ABB RAPID module: Module1.mod

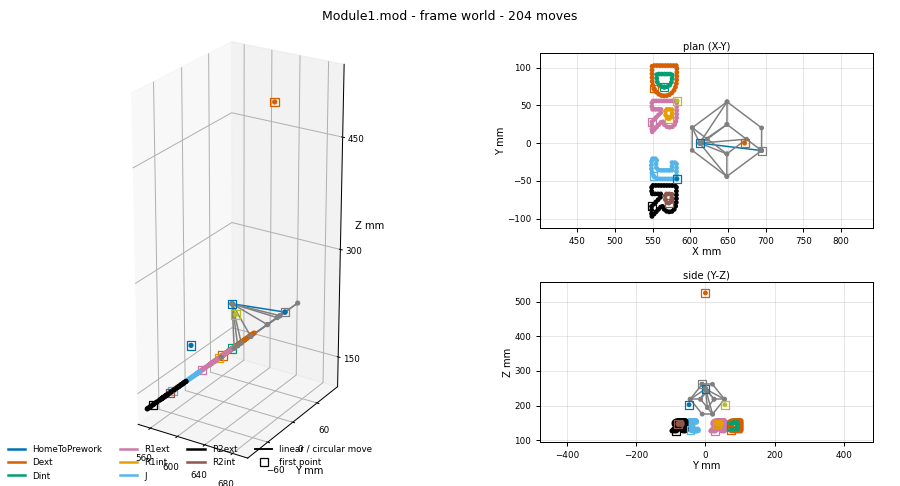
[picture p0: tool path of Module1.mod in frame world, 204 of 204 moves have a stored position in this frame; points joined in program order, loops and branches not executed]
MODULE Module1
    PERS tooldata MyNewTool:=[TRUE,[[40,0,140],[1,0,0,0]],[0.2,[0,0,1],[1,0,0,0],0,0,0]];
    PERS tooldata MaRCK:=[TRUE,[[40,0,140],[1,0,0,0]],[1,[0,0,60],[1,0,0,0],0,0,0]];
    PERS tooldata Marcket:=[TRUE,[[40,0,140],[1,0,0,0]],[1,[0,0,1],[1,0,0,0],0,0,0]];
    CONST robtarget PreworkLogo:=[[612.590636345,0.112352276,247.897245036],[0.173647946,0.001613761,0.984806431,-0.000284548],[-1,0,0,0],[9E+09,9E+09,9E+09,9E+09,9E+09,9E+09]];
    CONST robtarget EDext_10:=[[551.912875252,72.53519352,128.929412083],[0.173647946,0.001613761,0.984806431,-0.000284548],[0,-2,1,0],[9E+09,9E+09,9E+09,9E+09,9E+09,9E+09]];
    CONST robtarget EDext_20:=[[550.351593621,77.035190099,127.453730912],[0.173647946,0.001613761,0.984806431,-0.000284548],[0,0,0,0],[9E+09,9E+09,9E+09,9E+09,9E+09,9E+09]];
    CONST robtarget EDext_30:=[[549.633220287,81.925977855,126.766089465],[0.173647946,0.001613761,0.984806431,-0.000284548],[0,0,0,0],[9E+09,9E+09,9E+09,9E+09,9E+09,9E+09]];
    CONST robtarget EDext_40:=[[549.374310427,86.910926647,126.508367741],[0.173647946,0.001613761,0.984806431,-0.000284548],[0,0,0,0],[9E+09,9E+09,9E+09,9E+09,9E+09,9E+09]];
    CONST robtarget EDext_50:=[[549.36766375,91.910642603,126.486801869],[0.173647946,0.001613761,0.984806431,-0.000284548],[0,0,0,0],[9E+09,9E+09,9E+09,9E+09,9E+09,9E+09]];
    CONST robtarget EDext_60:=[[549.384050297,96.910615751,126.486801869],[0.173647946,0.001613761,0.984806431,-0.000284548],[0,0,0,0],[9E+09,9E+09,9E+09,9E+09,9E+09,9E+09]];
    CONST robtarget EDext_70:=[[549.400436844,101.910588899,126.486801869],[0.173647946,0.001613761,0.984806431,-0.000284548],[0,0,0,0],[9E+09,9E+09,9E+09,9E+09,9E+09,9E+09]];
    CONST robtarget EDext_80:=[[552.263411146,102.983965117,129.164192022],[0.173647946,0.001613761,0.984806431,-0.000284548],[0,0,0,0],[9E+09,9E+09,9E+09,9E+09,9E+09,9E+09]];
    CONST robtarget EDext_90:=[[555.913201428,102.97200356,132.581630802],[0.173647946,0.001613761,0.984806431,-0.000284548],[0,0,0,0],[9E+09,9E+09,9E+09,9E+09,9E+09,9E+09]];
    CONST robtarget EDext_100:=[[559.562991711,102.960042004,135.999069582],[0.173647946,0.001613761,0.984806431,-0.000284548],[0,0,0,0],[9E+09,9E+09,9E+09,9E+09,9E+09,9E+09]];
    CONST robtarget EDext_110:=[[563.212781993,102.948080447,139.416508362],[0.173647946,0.001613761,0.984806431,-0.000284548],[0,0,0,0],[9E+09,9E+09,9E+09,9E+09,9E+09,9E+09]];
    CONST robtarget EDext_120:=[[566.862572275,102.936118891,142.833947142],[0.173647946,0.001613761,0.984806431,-0.000284548],[0,0,0,0],[9E+09,9E+09,9E+09,9E+09,9E+09,9E+09]];
    CONST robtarget EDext_130:=[[570.512362558,102.924157334,146.251385922],[0.173647946,0.001613761,0.984806431,-0.000284548],[0,0,0,0],[9E+09,9E+09,9E+09,9E+09,9E+09,9E+09]];
    CONST robtarget EDext_140:=[[574.16215284,102.912195777,149.668824701],[0.173647946,0.001613761,0.984806431,-0.000284548],[0,0,0,0],[9E+09,9E+09,9E+09,9E+09,9E+09,9E+09]];
    CONST robtarget EDext_150:=[[577.811943123,102.900234221,153.086263481],[0.173647946,0.001613761,0.984806431,-0.000284548],[0,0,0,0],[9E+09,9E+09,9E+09,9E+09,9E+09,9E+09]];
    CONST robtarget EDext_160:=[[581.461733405,102.888272664,156.503702261],[0.173647946,0.001613761,0.984806431,-0.000284548],[0,0,0,0],[9E+09,9E+09,9E+09,9E+09,9E+09,9E+09]];
    CONST robtarget EDext_170:=[[582.239259874,98.968456724,157.243750889],[0.173647946,0.001613761,0.984806431,-0.000284548],[0,0,0,0],[9E+09,9E+09,9E+09,9E+09,9E+09,9E+09]];
    CONST robtarget EDext_180:=[[582.222873327,93.968483576,157.243750889],[0.173647946,0.001613761,0.984806431,-0.000284548],[0,0,0,0],[9E+09,9E+09,9E+09,9E+09,9E+09,9E+09]];
    CONST robtarget EDext_190:=[[582.206486779,88.968510428,157.243750889],[0.173647946,0.001613761,0.984806431,-0.000284548],[0,0,0,0],[9E+09,9E+09,9E+09,9E+09,9E+09,9E+09]];
    CONST robtarget EDext_200:=[[582.05998145,83.973285517,157.121902414],[0.173647946,0.001613761,0.984806431,-0.000284548],[0,0,0,0],[9E+09,9E+09,9E+09,9E+09,9E+09,9E+09]];
    CONST robtarget EDext_210:=[[581.599769178,79.014590704,156.706209142],[0.173647946,0.001613761,0.984806431,-0.000284548],[0,0,0,0],[9E+09,9E+09,9E+09,9E+09,9E+09,9E+09]];
    CONST robtarget EDext_220:=[[580.404388174,74.301796937,155.601401967],[0.173647946,0.001613761,0.984806431,-0.000284548],[0,0,0,0],[9E+09,9E+09,9E+09,9E+09,9E+09,9E+09]];
    CONST robtarget EDext_230:=[[578.391013182,70.140860724,153.728990378],[0.173647946,0.001613761,0.984806431,-0.000284548],[0,0,0,0],[9E+09,9E+09,9E+09,9E+09,9E+09,9E+09]];
    CONST robtarget EDext_240:=[[575.690696414,66.788466394,151.210894602],[0.173647946,0.001613761,0.984806431,-0.000284548],[0,0,0,0],[9E+09,9E+09,9E+09,9E+09,9E+09,9E+09]];
    CONST robtarget EDext_250:=[[572.487460802,64.407050959,148.218922062],[0.173647946,0.001613761,0.984806431,-0.000284548],[0,0,0,0],[9E+09,9E+09,9E+09,9E+09,9E+09,9E+09]];
    CONST robtarget EDext_260:=[[568.966787181,63.118163403,144.926370726],[0.173647946,0.001613761,0.984806431,-0.000284548],[0,0,0,0],[9E+09,9E+09,9E+09,9E+09,9E+09,9E+09]];
    CONST robtarget EDext_270:=[[565.328580893,62.794822032,141.520807298],[0.173647946,0.001613761,0.984806431,-0.000284548],[0,0,0,0],[9E+09,9E+09,9E+09,9E+09,9E+09,9E+09]];
    CONST robtarget EDext_280:=[[561.709530664,63.365475702,138.130436868],[0.173647946,0.001613761,0.984806431,-0.000284548],[0,0,0,0],[9E+09,9E+09,9E+09,9E+09,9E+09,9E+09]];
    CONST robtarget EDext_290:=[[558.268704982,64.989283235,134.903711368],[0.173647946,0.001613761,0.984806431,-0.000284548],[0,0,0,0],[9E+09,9E+09,9E+09,9E+09,9E+09,9E+09]];
    CONST robtarget EDext_300:=[[555.180659774,67.628712266,132.004187631],[0.173647946,0.001613761,0.984806431,-0.000284548],[0,0,0,0],[9E+09,9E+09,9E+09,9E+09,9E+09,9E+09]];
    CONST robtarget EDext_310:=[[552.613212389,71.156303357,129.589388927],[0.173647946,0.001613761,0.984806431,-0.000284548],[0,0,0,0],[9E+09,9E+09,9E+09,9E+09,9E+09,9E+09]];
    CONST robtarget FDint_10:=[[565.761082243,74.386090886,141.890200973],[0.173647946,0.001613761,0.984806431,-0.000284548],[0,-2,1,0],[9E+09,9E+09,9E+09,9E+09,9E+09,9E+09]];
    CONST robtarget FDint_20:=[[569.379445273,74.944551838,145.276463096],[0.173647946,0.001613761,0.984806431,-0.000284548],[0,0,0,0],[9E+09,9E+09,9E+09,9E+09,9E+09,9E+09]];
    CONST robtarget FDint_30:=[[572.681520952,77.008685984,148.361956019],[0.173647946,0.001613761,0.984806431,-0.000284548],[0,0,0,0],[9E+09,9E+09,9E+09,9E+09,9E+09,9E+09]];
    CONST robtarget FDint_40:=[[575.047866711,80.768438651,150.566095233],[0.173647946,0.001613761,0.984806431,-0.000284548],[0,0,0,0],[9E+09,9E+09,9E+09,9E+09,9E+09,9E+09]];
    CONST robtarget FDint_50:=[[575.986682219,85.560327407,151.430430149],[0.173647946,0.001613761,0.984806431,-0.000284548],[0,0,0,0],[9E+09,9E+09,9E+09,9E+09,9E+09,9E+09]];
    CONST robtarget FDint_60:=[[576.087876515,90.558290854,151.509844214],[0.173647946,0.001613761,0.984806431,-0.000284548],[0,0,0,0],[9E+09,9E+09,9E+09,9E+09,9E+09,9E+09]];
    CONST robtarget FDint_70:=[[573.20406064,91.610574886,148.806416589],[0.173647946,0.001613761,0.984806431,-0.000284548],[0,0,0,0],[9E+09,9E+09,9E+09,9E+09,9E+09,9E+09]];
    CONST robtarget FDint_80:=[[569.554270358,91.622536443,145.388977809],[0.173647946,0.001613761,0.984806431,-0.000284548],[0,0,0,0],[9E+09,9E+09,9E+09,9E+09,9E+09,9E+09]];
    CONST robtarget FDint_90:=[[565.904480074,91.634497999,141.971539029],[0.173647946,0.001613761,0.984806431,-0.000284548],[0,0,0,0],[9E+09,9E+09,9E+09,9E+09,9E+09,9E+09]];
    CONST robtarget FDint_100:=[[562.254689792,91.646459556,138.554100249],[0.173647946,0.001613761,0.984806431,-0.000284548],[0,0,0,0],[9E+09,9E+09,9E+09,9E+09,9E+09,9E+09]];
    CONST robtarget FDint_110:=[[558.604899509,91.658421112,135.136661469],[0.173647946,0.001613761,0.984806431,-0.000284548],[0,0,0,0],[9E+09,9E+09,9E+09,9E+09,9E+09,9E+09]];
    CONST robtarget FDint_120:=[[555.51395758,90.900193665,132.244851682],[0.173647946,0.001613761,0.984806431,-0.000284548],[0,0,0,0],[9E+09,9E+09,9E+09,9E+09,9E+09,9E+09]];
    CONST robtarget FDint_130:=[[555.56318478,85.901073737,132.306285076],[0.173647946,0.001613761,0.984806431,-0.000284548],[0,0,0,0],[9E+09,9E+09,9E+09,9E+09,9E+09,9E+09]];
    CONST robtarget FDint_140:=[[556.34730194,81.067926581,133.055307452],[0.173647946,0.001613761,0.984806431,-0.000284548],[0,0,0,0],[9E+09,9E+09,9E+09,9E+09,9E+09,9E+09]];
    CONST robtarget FDint_150:=[[558.624417237,77.220561783,135.199241268],[0.173647946,0.001613761,0.984806431,-0.000284548],[0,0,0,0],[9E+09,9E+09,9E+09,9E+09,9E+09,9E+09]];
    CONST robtarget FDint_160:=[[561.87847136,75.038381865,138.252800717],[0.173647946,0.001613761,0.984806431,-0.000284548],[0,0,0,0],[9E+09,9E+09,9E+09,9E+09,9E+09,9E+09]];
    CONST robtarget FDint_170:=[[565.486835279,74.389591817,141.633405025],[0.173647946,0.001613761,0.984806431,-0.000284548],[0,0,0,0],[9E+09,9E+09,9E+09,9E+09,9E+09,9E+09]];
    CONST robtarget GR1ext_10:=[[549.159222937,28.309785163,126.486801869],[0.173647946,0.001613761,0.984806431,-0.000284548],[0,0,0,0],[9E+09,9E+09,9E+09,9E+09,9E+09,9E+09]];
    CONST robtarget GR1ext_20:=[[552.078895967,31.318504465,129.211341749],[0.173647946,0.001613761,0.984806431,-0.000284548],[0,0,0,0],[9E+09,9E+09,9E+09,9E+09,9E+09,9E+09]];
    CONST robtarget GR1ext_30:=[[554.998568997,34.327223766,131.93588163],[0.173647946,0.001613761,0.984806431,-0.000284548],[0,0,0,0],[9E+09,9E+09,9E+09,9E+09,9E+09,9E+09]];
    CONST robtarget GR1ext_40:=[[557.918242027,37.335943068,134.660421511],[0.173647946,0.001613761,0.984806431,-0.000284548],[0,0,0,0],[9E+09,9E+09,9E+09,9E+09,9E+09,9E+09]];
    CONST robtarget GR1ext_50:=[[560.837915058,40.344662369,137.384961391],[0.173647946,0.001613761,0.984806431,-0.000284548],[0,0,0,0],[9E+09,9E+09,9E+09,9E+09,9E+09,9E+09]];
    CONST robtarget GR1ext_60:=[[561.129703813,44.863025586,137.644306177],[0.173647946,0.001613761,0.984806431,-0.000284548],[0,0,0,0],[9E+09,9E+09,9E+09,9E+09,9E+09,9E+09]];
    CONST robtarget GR1ext_70:=[[557.47991353,44.874987143,134.226867398],[0.173647946,0.001613761,0.984806431,-0.000284548],[0,0,0,0],[9E+09,9E+09,9E+09,9E+09,9E+09,9E+09]];
    CONST robtarget GR1ext_80:=[[553.830123248,44.886948699,130.809428618],[0.173647946,0.001613761,0.984806431,-0.000284548],[0,0,0,0],[9E+09,9E+09,9E+09,9E+09,9E+09,9E+09]];
    CONST robtarget GR1ext_90:=[[550.180332966,44.898910256,127.391989838],[0.173647946,0.001613761,0.984806431,-0.000284548],[0,0,0,0],[9E+09,9E+09,9E+09,9E+09,9E+09,9E+09]];
    CONST robtarget GR1ext_100:=[[549.2256475,48.577692778,126.486801869],[0.173647946,0.001613761,0.984806431,-0.000284548],[0,0,0,0],[9E+09,9E+09,9E+09,9E+09,9E+09,9E+09]];
    CONST robtarget GR1ext_110:=[[549.242034047,53.577665926,126.486801869],[0.173647946,0.001613761,0.984806431,-0.000284548],[0,0,0,0],[9E+09,9E+09,9E+09,9E+09,9E+09,9E+09]];
    CONST robtarget GR1ext_120:=[[551.034331948,56.127938354,128.157155282],[0.173647946,0.001613761,0.984806431,-0.000284548],[0,0,0,0],[9E+09,9E+09,9E+09,9E+09,9E+09,9E+09]];
    CONST robtarget GR1ext_130:=[[554.68412223,56.115976798,131.574594062],[0.173647946,0.001613761,0.984806431,-0.000284548],[0,0,0,0],[9E+09,9E+09,9E+09,9E+09,9E+09,9E+09]];
    CONST robtarget GR1ext_140:=[[558.333912513,56.104015241,134.992032842],[0.173647946,0.001613761,0.984806431,-0.000284548],[0,0,0,0],[9E+09,9E+09,9E+09,9E+09,9E+09,9E+09]];
    CONST robtarget GR1ext_150:=[[561.983702796,56.092053685,138.409471622],[0.173647946,0.001613761,0.984806431,-0.000284548],[0,0,0,0],[9E+09,9E+09,9E+09,9E+09,9E+09,9E+09]];
    CONST robtarget GR1ext_160:=[[565.633493078,56.080092128,141.826910402],[0.173647946,0.001613761,0.984806431,-0.000284548],[0,0,0,0],[9E+09,9E+09,9E+09,9E+09,9E+09,9E+09]];
    CONST robtarget GR1ext_170:=[[569.283283361,56.068130572,145.244349182],[0.173647946,0.001613761,0.984806431,-0.000284548],[0,0,0,0],[9E+09,9E+09,9E+09,9E+09,9E+09,9E+09]];
    CONST robtarget GR1ext_180:=[[572.933073643,56.056169015,148.661787962],[0.173647946,0.001613761,0.984806431,-0.000284548],[0,0,0,0],[9E+09,9E+09,9E+09,9E+09,9E+09,9E+09]];
    CONST robtarget GR1ext_190:=[[576.582863926,56.044207459,152.079226742],[0.173647946,0.001613761,0.984806431,-0.000284548],[0,0,0,0],[9E+09,9E+09,9E+09,9E+09,9E+09,9E+09]];
    CONST robtarget GR1ext_200:=[[580.232654208,56.032245902,155.496665522],[0.173647946,0.001613761,0.984806431,-0.000284548],[0,0,0,0],[9E+09,9E+09,9E+09,9E+09,9E+09,9E+09]];
    CONST robtarget GR1ext_210:=[[582.090514517,53.582276609,157.243750889],[0.173647946,0.001613761,0.984806431,-0.000284548],[0,0,0,0],[9E+09,9E+09,9E+09,9E+09,9E+09,9E+09]];
    CONST robtarget GR1ext_220:=[[582.07412797,48.582303461,157.243750889],[0.173647946,0.001613761,0.984806431,-0.000284548],[0,0,0,0],[9E+09,9E+09,9E+09,9E+09,9E+09,9E+09]];
    CONST robtarget GR1ext_230:=[[582.057741422,43.582330312,157.243750889],[0.173647946,0.001613761,0.984806431,-0.000284548],[0,0,0,0],[9E+09,9E+09,9E+09,9E+09,9E+09,9E+09]];
    CONST robtarget GR1ext_240:=[[582.041354875,38.582357164,157.243750889],[0.173647946,0.001613761,0.984806431,-0.000284548],[0,0,0,0],[9E+09,9E+09,9E+09,9E+09,9E+09,9E+09]];
    CONST robtarget GR1ext_250:=[[581.887031,33.588566956,157.114577286],[0.173647946,0.001613761,0.984806431,-0.000284548],[0,0,0,0],[9E+09,9E+09,9E+09,9E+09,9E+09,9E+09]];
    CONST robtarget GR1ext_260:=[[581.128662004,28.711829147,156.419459926],[0.173647946,0.001613761,0.984806431,-0.000284548],[0,0,0,0],[9E+09,9E+09,9E+09,9E+09,9E+09,9E+09]];
    CONST robtarget GR1ext_270:=[[579.222937052,24.480084612,154.648061408],[0.173647946,0.001613761,0.984806431,-0.000284548],[0,0,0,0],[9E+09,9E+09,9E+09,9E+09,9E+09,9E+09]];
    CONST robtarget GR1ext_280:=[[576.214714314,21.722189391,151.839840233],[0.173647946,0.001613761,0.984806431,-0.000284548],[0,0,0,0],[9E+09,9E+09,9E+09,9E+09,9E+09,9E+09]];
    CONST robtarget GR1ext_290:=[[572.616939057,21.053869541,148.473192144],[0.173647946,0.001613761,0.984806431,-0.000284548],[0,0,0,0],[9E+09,9E+09,9E+09,9E+09,9E+09,9E+09]];
    CONST robtarget GR1ext_300:=[[569.03162427,21.867677864,145.113663007],[0.173647946,0.001613761,0.984806431,-0.000284548],[0,0,0,0],[9E+09,9E+09,9E+09,9E+09,9E+09,9E+09]];
    CONST robtarget GR1ext_310:=[[565.933301553,24.431725119,142.204747469],[0.173647946,0.001613761,0.984806431,-0.000284548],[0,0,0,0],[9E+09,9E+09,9E+09,9E+09,9E+09,9E+09]];
    CONST robtarget GR1ext_320:=[[563.657751182,28.309232507,140.062186439],[0.173647946,0.001613761,0.984806431,-0.000284548],[0,0,0,0],[9E+09,9E+09,9E+09,9E+09,9E+09,9E+09]];
    CONST robtarget GR1ext_330:=[[561.138391327,27.497607501,137.705729007],[0.173647946,0.001613761,0.984806431,-0.000284548],[0,0,0,0],[9E+09,9E+09,9E+09,9E+09,9E+09,9E+09]];
    CONST robtarget GR1ext_340:=[[558.264968647,24.406364665,135.024747876],[0.173647946,0.001613761,0.984806431,-0.000284548],[0,0,0,0],[9E+09,9E+09,9E+09,9E+09,9E+09,9E+09]];
    CONST robtarget GR1ext_350:=[[555.391545966,21.315121829,132.343766744],[0.173647946,0.001613761,0.984806431,-0.000284548],[0,0,0,0],[9E+09,9E+09,9E+09,9E+09,9E+09,9E+09]];
    CONST robtarget GR1ext_360:=[[552.518123285,18.223878993,129.662785613],[0.173647946,0.001613761,0.984806431,-0.000284548],[0,0,0,0],[9E+09,9E+09,9E+09,9E+09,9E+09,9E+09]];
    CONST robtarget GR1ext_370:=[[549.644700604,15.132636157,126.981804481],[0.173647946,0.001613761,0.984806431,-0.000284548],[0,0,0,0],[9E+09,9E+09,9E+09,9E+09,9E+09,9E+09]];
    CONST robtarget GR1ext_380:=[[549.127527591,18.638688665,126.486801869],[0.173647946,0.001613761,0.984806431,-0.000284548],[0,0,0,0],[9E+09,9E+09,9E+09,9E+09,9E+09,9E+09]];
    CONST robtarget GR1ext_390:=[[549.143914138,23.638661813,126.486801869],[0.173647946,0.001613761,0.984806431,-0.000284548],[0,0,0,0],[9E+09,9E+09,9E+09,9E+09,9E+09,9E+09]];
    CONST robtarget HR1int_10:=[[571.959732893,32.647563873,147.822254349],[0.173647946,0.001613761,0.984806431,-0.000284548],[0,-2,1,0],[9E+09,9E+09,9E+09,9E+09,9E+09,9E+09]];
    CONST robtarget HR1int_20:=[[575.149419403,34.61134025,150.802822071],[0.173647946,0.001613761,0.984806431,-0.000284548],[0,0,0,0],[9E+09,9E+09,9E+09,9E+09,9E+09,9E+09]];
    CONST robtarget HR1int_30:=[[575.982626554,39.413197479,151.5682423],[0.173647946,0.001613761,0.984806431,-0.000284548],[0,0,0,0],[9E+09,9E+09,9E+09,9E+09,9E+09,9E+09]];
    CONST robtarget HR1int_40:=[[576.017836302,44.412828089,151.585868046],[0.173647946,0.001613761,0.984806431,-0.000284548],[0,0,0,0],[9E+09,9E+09,9E+09,9E+09,9E+09,9E+09]];
    CONST robtarget HR1int_50:=[[572.662368207,44.825229273,148.442782661],[0.173647946,0.001613761,0.984806431,-0.000284548],[0,0,0,0],[9E+09,9E+09,9E+09,9E+09,9E+09,9E+09]];
    CONST robtarget HR1int_60:=[[569.012577925,44.83719083,145.025343881],[0.173647946,0.001613761,0.984806431,-0.000284548],[0,0,0,0],[9E+09,9E+09,9E+09,9E+09,9E+09,9E+09]];
    CONST robtarget HR1int_70:=[[567.17340627,42.351576284,143.310902832],[0.173647946,0.001613761,0.984806431,-0.000284548],[0,0,0,0],[9E+09,9E+09,9E+09,9E+09,9E+09,9E+09]];
    CONST robtarget HR1int_80:=[[567.402598455,37.370563966,143.540786974],[0.173647946,0.001613761,0.984806431,-0.000284548],[0,0,0,0],[9E+09,9E+09,9E+09,9E+09,9E+09,9E+09]];
    CONST robtarget HR1int_90:=[[569.422495165,33.396346001,145.444269007],[0.173647946,0.001613761,0.984806431,-0.000284548],[0,0,0,0],[9E+09,9E+09,9E+09,9E+09,9E+09,9E+09]];
    CONST robtarget IJ_10:=[[551.320468068,-43.245490091,128.730015331],[0.173647946,0.001613761,0.984806431,-0.000284548],[0,0,0,0],[9E+09,9E+09,9E+09,9E+09,9E+09,9E+09]];
    CONST robtarget IJ_20:=[[549.426005203,-39.008514231,126.943174249],[0.173647946,0.001613761,0.984806431,-0.000284548],[0,0,0,0],[9E+09,9E+09,9E+09,9E+09,9E+09,9E+09]];
    CONST robtarget IJ_30:=[[548.586005622,-34.15957373,126.141779114],[0.173647946,0.001613761,0.984806431,-0.000284548],[0,0,0,0],[9E+09,9E+09,9E+09,9E+09,9E+09,9E+09]];
    CONST robtarget IJ_40:=[[548.477427418,-29.166511841,126.024792284],[0.173647946,0.001613761,0.984806431,-0.000284548],[0,0,0,0],[9E+09,9E+09,9E+09,9E+09,9E+09,9E+09]];
    CONST robtarget IJ_50:=[[548.710119201,-24.177436392,126.227358447],[0.173647946,0.001613761,0.984806431,-0.000284548],[0,0,0,0],[9E+09,9E+09,9E+09,9E+09,9E+09,9E+09]];
    CONST robtarget IJ_60:=[[550.104401144,-20.559048954,127.521760564],[0.173647946,0.001613761,0.984806431,-0.000284548],[0,0,0,0],[9E+09,9E+09,9E+09,9E+09,9E+09,9E+09]];
    CONST robtarget IJ_70:=[[553.754191426,-20.57101051,130.939199344],[0.173647946,0.001613761,0.984806431,-0.000284548],[0,0,0,0],[9E+09,9E+09,9E+09,9E+09,9E+09,9E+09]];
    CONST robtarget IJ_80:=[[555.465361118,-22.711275868,132.547983754],[0.173647946,0.001613761,0.984806431,-0.000284548],[0,0,0,0],[9E+09,9E+09,9E+09,9E+09,9E+09,9E+09]];
    CONST robtarget IJ_90:=[[554.680121136,-27.565791663,131.827638136],[0.173647946,0.001613761,0.984806431,-0.000284548],[0,0,0,0],[9E+09,9E+09,9E+09,9E+09,9E+09,9E+09]];
    CONST robtarget IJ_100:=[[555.145862124,-32.487268808,132.278826933],[0.173647946,0.001613761,0.984806431,-0.000284548],[0,0,0,0],[9E+09,9E+09,9E+09,9E+09,9E+09,9E+09]];
    CONST robtarget IJ_110:=[[557.841723431,-35.563111404,134.812476972],[0.173647946,0.001613761,0.984806431,-0.000284548],[0,0,0,0],[9E+09,9E+09,9E+09,9E+09,9E+09,9E+09]];
    CONST robtarget IJ_120:=[[561.46746702,-35.976374681,138.208631607],[0.173647946,0.001613761,0.984806431,-0.000284548],[0,0,0,0],[9E+09,9E+09,9E+09,9E+09,9E+09,9E+09]];
    CONST robtarget IJ_130:=[[565.117207108,-35.997312406,141.626050933],[0.173647946,0.001613761,0.984806431,-0.000284548],[0,0,0,0],[9E+09,9E+09,9E+09,9E+09,9E+09,9E+09]];
    CONST robtarget IJ_140:=[[568.766997391,-36.009273962,145.043489713],[0.173647946,0.001613761,0.984806431,-0.000284548],[0,0,0,0],[9E+09,9E+09,9E+09,9E+09,9E+09,9E+09]];
    CONST robtarget IJ_150:=[[572.416787673,-36.021235519,148.460928493],[0.173647946,0.001613761,0.984806431,-0.000284548],[0,0,0,0],[9E+09,9E+09,9E+09,9E+09,9E+09,9E+09]];
    CONST robtarget IJ_160:=[[575.835093356,-35.713886099,151.660641828],[0.173647946,0.001613761,0.984806431,-0.000284548],[0,0,0,0],[9E+09,9E+09,9E+09,9E+09,9E+09,9E+09]];
    CONST robtarget IJ_170:=[[575.851479904,-30.713912951,151.660641828],[0.173647946,0.001613761,0.984806431,-0.000284548],[0,0,0,0],[9E+09,9E+09,9E+09,9E+09,9E+09,9E+09]];
    CONST robtarget IJ_180:=[[575.893242248,-25.7489433,151.68450932],[0.173647946,0.001613761,0.984806431,-0.000284548],[0,0,0,0],[9E+09,9E+09,9E+09,9E+09,9E+09,9E+09]];
    CONST robtarget IJ_190:=[[579.543032531,-25.760904857,155.1019481],[0.173647946,0.001613761,0.984806431,-0.000284548],[0,0,0,0],[9E+09,9E+09,9E+09,9E+09,9E+09,9E+09]];
    CONST robtarget IJ_200:=[[581.824339743,-27.634754078,157.243750889],[0.173647946,0.001613761,0.984806431,-0.000284548],[0,0,0,0],[9E+09,9E+09,9E+09,9E+09,9E+09,9E+09]];
    CONST robtarget IJ_210:=[[581.807953196,-32.634727226,157.243750889],[0.173647946,0.001613761,0.984806431,-0.000284548],[0,0,0,0],[9E+09,9E+09,9E+09,9E+09,9E+09,9E+09]];
    CONST robtarget IJ_220:=[[581.791566648,-37.634700374,157.243750889],[0.173647946,0.001613761,0.984806431,-0.000284548],[0,0,0,0],[9E+09,9E+09,9E+09,9E+09,9E+09,9E+09]];
    CONST robtarget IJ_230:=[[581.775180101,-42.634673522,157.243750889],[0.173647946,0.001613761,0.984806431,-0.000284548],[0,0,0,0],[9E+09,9E+09,9E+09,9E+09,9E+09,9E+09]];
    CONST robtarget IJ_240:=[[581.556753069,-47.355951048,157.053719437],[0.173647946,0.001613761,0.984806431,-0.000284548],[0,0,0,0],[9E+09,9E+09,9E+09,9E+09,9E+09,9E+09]];
    CONST robtarget IJ_250:=[[577.906962787,-47.343989491,153.636280657],[0.173647946,0.001613761,0.984806431,-0.000284548],[0,0,0,0],[9E+09,9E+09,9E+09,9E+09,9E+09,9E+09]];
    CONST robtarget IJ_260:=[[574.257172505,-47.332027935,150.218841877],[0.173647946,0.001613761,0.984806431,-0.000284548],[0,0,0,0],[9E+09,9E+09,9E+09,9E+09,9E+09,9E+09]];
    CONST robtarget IJ_270:=[[570.607382222,-47.320066378,146.801403097],[0.173647946,0.001613761,0.984806431,-0.000284548],[0,0,0,0],[9E+09,9E+09,9E+09,9E+09,9E+09,9E+09]];
    CONST robtarget IJ_280:=[[566.95759194,-47.308104822,143.383964317],[0.173647946,0.001613761,0.984806431,-0.000284548],[0,0,0,0],[9E+09,9E+09,9E+09,9E+09,9E+09,9E+09]];
    CONST robtarget IJ_290:=[[563.307801657,-47.296143265,139.966525537],[0.173647946,0.001613761,0.984806431,-0.000284548],[0,0,0,0],[9E+09,9E+09,9E+09,9E+09,9E+09,9E+09]];
    CONST robtarget IJ_300:=[[559.658011375,-47.284181709,136.549086757],[0.173647946,0.001613761,0.984806431,-0.000284548],[0,0,0,0],[9E+09,9E+09,9E+09,9E+09,9E+09,9E+09]];
    CONST robtarget IJ_310:=[[556.029645572,-46.895903687,133.15055354],[0.173647946,0.001613761,0.984806431,-0.000284548],[0,0,0,0],[9E+09,9E+09,9E+09,9E+09,9E+09,9E+09]];
    CONST robtarget IJ_320:=[[552.702794125,-44.926549268,130.029484981],[0.173647946,0.001613761,0.984806431,-0.000284548],[0,0,0,0],[9E+09,9E+09,9E+09,9E+09,9E+09,9E+09]];
    CONST robtarget JR2ext_10:=[[548.791720768,-83.824939488,126.486801869],[0.173647946,0.001613761,0.984806431,-0.000284548],[0,0,0,0],[9E+09,9E+09,9E+09,9E+09,9E+09,9E+09]];
    CONST robtarget JR2ext_20:=[[551.711393798,-80.816220187,129.211341749],[0.173647946,0.001613761,0.984806431,-0.000284548],[0,0,0,0],[9E+09,9E+09,9E+09,9E+09,9E+09,9E+09]];
    CONST robtarget JR2ext_30:=[[554.631066828,-77.807500885,131.93588163],[0.173647946,0.001613761,0.984806431,-0.000284548],[0,0,0,0],[9E+09,9E+09,9E+09,9E+09,9E+09,9E+09]];
    CONST robtarget JR2ext_40:=[[557.550739858,-74.798781584,134.660421511],[0.173647946,0.001613761,0.984806431,-0.000284548],[0,0,0,0],[9E+09,9E+09,9E+09,9E+09,9E+09,9E+09]];
    CONST robtarget JR2ext_50:=[[560.470412889,-71.790062282,137.384961391],[0.173647946,0.001613761,0.984806431,-0.000284548],[0,0,0,0],[9E+09,9E+09,9E+09,9E+09,9E+09,9E+09]];
    CONST robtarget JR2ext_60:=[[560.762201643,-67.271699065,137.644306177],[0.173647946,0.001613761,0.984806431,-0.000284548],[0,0,0,0],[9E+09,9E+09,9E+09,9E+09,9E+09,9E+09]];
    CONST robtarget JR2ext_70:=[[557.11241136,-67.259737508,134.226867398],[0.173647946,0.001613761,0.984806431,-0.000284548],[0,0,0,0],[9E+09,9E+09,9E+09,9E+09,9E+09,9E+09]];
    CONST robtarget JR2ext_80:=[[553.462621078,-67.247775952,130.809428618],[0.173647946,0.001613761,0.984806431,-0.000284548],[0,0,0,0],[9E+09,9E+09,9E+09,9E+09,9E+09,9E+09]];
    CONST robtarget JR2ext_90:=[[549.812830796,-67.235814395,127.391989838],[0.173647946,0.001613761,0.984806431,-0.000284548],[0,0,0,0],[9E+09,9E+09,9E+09,9E+09,9E+09,9E+09]];
    CONST robtarget JR2ext_100:=[[548.85814533,-63.557031873,126.486801869],[0.173647946,0.001613761,0.984806431,-0.000284548],[0,0,0,0],[9E+09,9E+09,9E+09,9E+09,9E+09,9E+09]];
    CONST robtarget JR2ext_110:=[[548.874531877,-58.557058725,126.486801869],[0.173647946,0.001613761,0.984806431,-0.000284548],[0,0,0,0],[9E+09,9E+09,9E+09,9E+09,9E+09,9E+09]];
    CONST robtarget JR2ext_120:=[[550.666829779,-56.006786298,128.157155282],[0.173647946,0.001613761,0.984806431,-0.000284548],[0,0,0,0],[9E+09,9E+09,9E+09,9E+09,9E+09,9E+09]];
    CONST robtarget JR2ext_130:=[[554.316620061,-56.018747854,131.574594062],[0.173647946,0.001613761,0.984806431,-0.000284548],[0,0,0,0],[9E+09,9E+09,9E+09,9E+09,9E+09,9E+09]];
    CONST robtarget JR2ext_140:=[[557.966410343,-56.030709411,134.992032842],[0.173647946,0.001613761,0.984806431,-0.000284548],[0,0,0,0],[9E+09,9E+09,9E+09,9E+09,9E+09,9E+09]];
    CONST robtarget JR2ext_150:=[[561.616200626,-56.042670968,138.409471622],[0.173647946,0.001613761,0.984806431,-0.000284548],[0,0,0,0],[9E+09,9E+09,9E+09,9E+09,9E+09,9E+09]];
    CONST robtarget JR2ext_160:=[[565.265990908,-56.054632524,141.826910402],[0.173647946,0.001613761,0.984806431,-0.000284548],[0,0,0,0],[9E+09,9E+09,9E+09,9E+09,9E+09,9E+09]];
    CONST robtarget JR2ext_170:=[[568.915781191,-56.066594081,145.244349182],[0.173647946,0.001613761,0.984806431,-0.000284548],[0,0,0,0],[9E+09,9E+09,9E+09,9E+09,9E+09,9E+09]];
    CONST robtarget JR2ext_180:=[[572.565571473,-56.078555637,148.661787962],[0.173647946,0.001613761,0.984806431,-0.000284548],[0,0,0,0],[9E+09,9E+09,9E+09,9E+09,9E+09,9E+09]];
    CONST robtarget JR2ext_190:=[[576.215361756,-56.090517194,152.079226742],[0.173647946,0.001613761,0.984806431,-0.000284548],[0,0,0,0],[9E+09,9E+09,9E+09,9E+09,9E+09,9E+09]];
    CONST robtarget JR2ext_200:=[[579.865152038,-56.10247875,155.496665522],[0.173647946,0.001613761,0.984806431,-0.000284548],[0,0,0,0],[9E+09,9E+09,9E+09,9E+09,9E+09,9E+09]];
    CONST robtarget JR2ext_210:=[[581.723012347,-58.552448044,157.243750889],[0.173647946,0.001613761,0.984806431,-0.000284548],[0,0,0,0],[9E+09,9E+09,9E+09,9E+09,9E+09,9E+09]];
    CONST robtarget JR2ext_220:=[[581.7066258,-63.552421192,157.243750889],[0.173647946,0.001613761,0.984806431,-0.000284548],[0,0,0,0],[9E+09,9E+09,9E+09,9E+09,9E+09,9E+09]];
    CONST robtarget JR2ext_230:=[[581.690239253,-68.55239434,157.243750889],[0.173647946,0.001613761,0.984806431,-0.000284548],[0,0,0,0],[9E+09,9E+09,9E+09,9E+09,9E+09,9E+09]];
    CONST robtarget JR2ext_240:=[[581.673852705,-73.552367488,157.243750889],[0.173647946,0.001613761,0.984806431,-0.000284548],[0,0,0,0],[9E+09,9E+09,9E+09,9E+09,9E+09,9E+09]];
    CONST robtarget JR2ext_250:=[[581.51952883,-78.546157695,157.114577286],[0.173647946,0.001613761,0.984806431,-0.000284548],[0,0,0,0],[9E+09,9E+09,9E+09,9E+09,9E+09,9E+09]];
    CONST robtarget JR2ext_260:=[[580.761159835,-83.422895504,156.419459926],[0.173647946,0.001613761,0.984806431,-0.000284548],[0,0,0,0],[9E+09,9E+09,9E+09,9E+09,9E+09,9E+09]];
    CONST robtarget JR2ext_270:=[[578.855434883,-87.654640039,154.648061408],[0.173647946,0.001613761,0.984806431,-0.000284548],[0,0,0,0],[9E+09,9E+09,9E+09,9E+09,9E+09,9E+09]];
    CONST robtarget JR2ext_280:=[[575.847212144,-90.41253526,151.839840233],[0.173647946,0.001613761,0.984806431,-0.000284548],[0,0,0,0],[9E+09,9E+09,9E+09,9E+09,9E+09,9E+09]];
    CONST robtarget JR2ext_290:=[[572.249436888,-91.08085511,148.473192144],[0.173647946,0.001613761,0.984806431,-0.000284548],[0,0,0,0],[9E+09,9E+09,9E+09,9E+09,9E+09,9E+09]];
    CONST robtarget JR2ext_300:=[[568.664122101,-90.267046787,145.113663007],[0.173647946,0.001613761,0.984806431,-0.000284548],[0,0,0,0],[9E+09,9E+09,9E+09,9E+09,9E+09,9E+09]];
    CONST robtarget JR2ext_310:=[[565.565799383,-87.702999533,142.204747469],[0.173647946,0.001613761,0.984806431,-0.000284548],[0,0,0,0],[9E+09,9E+09,9E+09,9E+09,9E+09,9E+09]];
    CONST robtarget JR2ext_320:=[[563.290249012,-83.825492144,140.062186439],[0.173647946,0.001613761,0.984806431,-0.000284548],[0,0,0,0],[9E+09,9E+09,9E+09,9E+09,9E+09,9E+09]];
    CONST robtarget JR2ext_330:=[[560.770889158,-84.637117152,137.705729007],[0.173647946,0.001613761,0.984806431,-0.000284548],[0,0,0,0],[9E+09,9E+09,9E+09,9E+09,9E+09,9E+09]];
    CONST robtarget JR2ext_340:=[[557.897466477,-87.728359987,135.024747876],[0.173647946,0.001613761,0.984806431,-0.000284548],[0,0,0,0],[9E+09,9E+09,9E+09,9E+09,9E+09,9E+09]];
    CONST robtarget JR2ext_350:=[[555.024043796,-90.819602822,132.343766744],[0.173647946,0.001613761,0.984806431,-0.000284548],[0,0,0,0],[9E+09,9E+09,9E+09,9E+09,9E+09,9E+09]];
    CONST robtarget JR2ext_360:=[[552.150621115,-93.910845658,129.662785613],[0.173647946,0.001613761,0.984806431,-0.000284548],[0,0,0,0],[9E+09,9E+09,9E+09,9E+09,9E+09,9E+09]];
    CONST robtarget JR2ext_370:=[[549.277198434,-97.002088494,126.981804481],[0.173647946,0.001613761,0.984806431,-0.000284548],[0,0,0,0],[9E+09,9E+09,9E+09,9E+09,9E+09,9E+09]];
    CONST robtarget JR2ext_380:=[[548.760025421,-93.496035986,126.486801869],[0.173647946,0.001613761,0.984806431,-0.000284548],[0,0,0,0],[9E+09,9E+09,9E+09,9E+09,9E+09,9E+09]];
    CONST robtarget JR2ext_390:=[[548.776411969,-88.496062838,126.486801869],[0.173647946,0.001613761,0.984806431,-0.000284548],[0,0,0,0],[9E+09,9E+09,9E+09,9E+09,9E+09,9E+09]];
    CONST robtarget KR2int_10:=[[571.592230724,-79.487160779,147.822254349],[0.173647946,0.001613761,0.984806431,-0.000284548],[0,0,0,0],[9E+09,9E+09,9E+09,9E+09,9E+09,9E+09]];
    CONST robtarget KR2int_20:=[[574.781917233,-77.523384401,150.802822071],[0.173647946,0.001613761,0.984806431,-0.000284548],[0,0,0,0],[9E+09,9E+09,9E+09,9E+09,9E+09,9E+09]];
    CONST robtarget KR2int_30:=[[575.615124384,-72.721527172,151.5682423],[0.173647946,0.001613761,0.984806431,-0.000284548],[0,0,0,0],[9E+09,9E+09,9E+09,9E+09,9E+09,9E+09]];
    CONST robtarget KR2int_40:=[[575.650334132,-67.721896562,151.585868046],[0.173647946,0.001613761,0.984806431,-0.000284548],[0,0,0,0],[9E+09,9E+09,9E+09,9E+09,9E+09,9E+09]];
    CONST robtarget KR2int_50:=[[572.294866037,-67.309495378,148.442782661],[0.173647946,0.001613761,0.984806431,-0.000284548],[0,0,0,0],[9E+09,9E+09,9E+09,9E+09,9E+09,9E+09]];
    CONST robtarget KR2int_60:=[[568.645075755,-67.297533822,145.025343881],[0.173647946,0.001613761,0.984806431,-0.000284548],[0,0,0,0],[9E+09,9E+09,9E+09,9E+09,9E+09,9E+09]];
    CONST robtarget KR2int_70:=[[566.8059041,-69.783148368,143.310902832],[0.173647946,0.001613761,0.984806431,-0.000284548],[0,0,0,0],[9E+09,9E+09,9E+09,9E+09,9E+09,9E+09]];
    CONST robtarget KR2int_80:=[[567.035096285,-74.764160685,143.540786974],[0.173647946,0.001613761,0.984806431,-0.000284548],[0,0,0,0],[9E+09,9E+09,9E+09,9E+09,9E+09,9E+09]];
    CONST robtarget KR2int_90:=[[569.054992995,-78.73837865,145.444269007],[0.173647946,0.001613761,0.984806431,-0.000284548],[0,0,0,0],[9E+09,9E+09,9E+09,9E+09,9E+09,9E+09]];
    CONST robtarget RA:=[[694.598675159,-9.776467715,261.412261981],[0.173647946,0.001613761,0.984806431,-0.000284548],[0,0,0,0],[9E+09,9E+09,9E+09,9E+09,9E+09,9E+09]];
    CONST robtarget RB:=[[694.696994443,20.223371173,261.412261981],[0.173647946,0.001613761,0.984806431,-0.000284548],[0,0,0,0],[9E+09,9E+09,9E+09,9E+09,9E+09,9E+09]];
    CONST robtarget RC:=[[648.822308594,54.873902803,218.353261981],[0.173647946,0.001613761,0.984806431,-0.000284548],[0,0,0,0],[9E+09,9E+09,9E+09,9E+09,9E+09,9E+09]];
    CONST robtarget RD:=[[602.722488385,20.524801712,175.293261981],[0.173647946,0.001613761,0.984806431,-0.000284548],[-1,0,0,0],[9E+09,9E+09,9E+09,9E+09,9E+09,9E+09]];
    CONST robtarget RE:=[[602.624169101,-9.475037176,175.293261981],[0.173647946,0.001613761,0.984806431,-0.000284548],[-1,0,0,0],[9E+09,9E+09,9E+09,9E+09,9E+09,9E+09]];
    CONST robtarget RF:=[[648.497854955,-44.125565528,218.353261981],[0.173647946,0.001613761,0.984806431,-0.000284548],[-1,0,0,0],[9E+09,9E+09,9E+09,9E+09,9E+09,9E+09]];
    CONST robtarget RH:=[[648.723989309,24.874063915,218.353261981],[0.173647946,0.001613761,0.984806431,-0.000284548],[-1,0,0,0],[9E+09,9E+09,9E+09,9E+09,9E+09,9E+09]];
    CONST robtarget RI:=[[622.667221367,5.459355743,194.015261981],[0.173647946,0.001613761,0.984806431,-0.000284548],[-1,0,0,0],[9E+09,9E+09,9E+09,9E+09,9E+09,9E+09]];
    CONST robtarget RJ:=[[648.59617424,-14.12572664,218.353261981],[0.173647946,0.001613761,0.984806431,-0.000284548],[-1,0,0,0],[9E+09,9E+09,9E+09,9E+09,9E+09,9E+09]];
    CONST robtarget RG:=[[674.652942182,5.288981532,242.691261981],[0.173647946,0.001613761,0.984806431,-0.000284548],[-1,0,0,0],[9E+09,9E+09,9E+09,9E+09,9E+09,9E+09]];
    CONST robtarget PreworkDR:=[[582.781724283,56.024344414,202.514261981],[0.173647946,0.001613761,0.984806431,-0.000284548],[0,0,0,0],[9E+09,9E+09,9E+09,9E+09,9E+09,9E+09]];
    CONST robtarget PreworkJR:=[[582.44290292,-47.359100373,202.514261981],[0.173647946,0.001613761,0.984806431,-0.000284548],[0,0,0,0],[9E+09,9E+09,9E+09,9E+09,9E+09,9E+09]];
    CONST robtarget MHomeIntermed:=[[672.102434247,-0.055687782,525.015369008],[0.173647946,0.001613761,0.984806431,-0.000284548],[0,-2,1,0],[9E+09,9E+09,9E+09,9E+09,9E+09,9E+09]];
    PROC HomeToPrework()
        MoveL PreworkLogo,v1000,z100,Marcket\WObj:=wobj0;
        MoveL RA,v500,fine,Marcket\WObj:=wobj0;

    ENDPROC
    PROC Dext()
        MoveL EDext_10,v500,z100,Marcket\WObj:=wobj0;
        MoveL EDext_20,v500,z100,Marcket\WObj:=wobj0;
        MoveL EDext_30,v500,z100,Marcket\WObj:=wobj0;
        MoveL EDext_40,v500,z100,Marcket\WObj:=wobj0;
        MoveL EDext_50,v500,z100,Marcket\WObj:=wobj0;
        MoveL EDext_60,v500,z100,Marcket\WObj:=wobj0;
        MoveL EDext_70,v500,z100,Marcket\WObj:=wobj0;
        MoveL EDext_80,v500,z100,Marcket\WObj:=wobj0;
        MoveL EDext_90,v500,z100,Marcket\WObj:=wobj0;
        MoveL EDext_100,v500,z100,Marcket\WObj:=wobj0;
        MoveL EDext_110,v500,z100,Marcket\WObj:=wobj0;
        MoveL EDext_120,v500,z100,Marcket\WObj:=wobj0;
        MoveL EDext_130,v500,z100,Marcket\WObj:=wobj0;
        MoveL EDext_140,v500,z100,Marcket\WObj:=wobj0;
        MoveL EDext_150,v500,z100,Marcket\WObj:=wobj0;
        MoveL EDext_160,v500,z100,Marcket\WObj:=wobj0;
        MoveL EDext_170,v500,z100,Marcket\WObj:=wobj0;
        MoveL EDext_180,v500,z100,Marcket\WObj:=wobj0;
        MoveL EDext_190,v500,z100,Marcket\WObj:=wobj0;
        MoveL EDext_200,v500,z100,Marcket\WObj:=wobj0;
        MoveL EDext_210,v500,z100,Marcket\WObj:=wobj0;
        MoveL EDext_220,v500,z100,Marcket\WObj:=wobj0;
        MoveL EDext_230,v500,z100,Marcket\WObj:=wobj0;
        MoveL EDext_240,v500,z100,Marcket\WObj:=wobj0;
        MoveL EDext_250,v500,z100,Marcket\WObj:=wobj0;
        MoveL EDext_260,v500,z100,Marcket\WObj:=wobj0;
        MoveL EDext_270,v500,z100,Marcket\WObj:=wobj0;
        MoveL EDext_280,v500,z100,Marcket\WObj:=wobj0;
        MoveL EDext_290,v500,z100,Marcket\WObj:=wobj0;
        MoveL EDext_300,v500,z100,Marcket\WObj:=wobj0;
        MoveL EDext_310,v500,z100,Marcket\WObj:=wobj0;
        MoveL EDext_10,v500,z100,Marcket\WObj:=wobj0;

    ENDPROC
    PROC Dint()
        MoveL FDint_10,v500,z100,Marcket\WObj:=wobj0;
        MoveL FDint_20,v500,z100,Marcket\WObj:=wobj0;
        MoveL FDint_30,v500,z100,Marcket\WObj:=wobj0;
        MoveL FDint_40,v500,z100,Marcket\WObj:=wobj0;
        MoveL FDint_50,v500,z100,Marcket\WObj:=wobj0;
        MoveL FDint_60,v500,z100,Marcket\WObj:=wobj0;
        MoveL FDint_70,v500,z100,Marcket\WObj:=wobj0;
        MoveL FDint_80,v500,z100,Marcket\WObj:=wobj0;
        MoveL FDint_90,v500,z100,Marcket\WObj:=wobj0;
        MoveL FDint_100,v500,z100,Marcket\WObj:=wobj0;
        MoveL FDint_110,v500,z100,Marcket\WObj:=wobj0;
        MoveL FDint_120,v500,z100,Marcket\WObj:=wobj0;
        MoveL FDint_130,v500,z100,Marcket\WObj:=wobj0;
        MoveL FDint_140,v500,z100,Marcket\WObj:=wobj0;
        MoveL FDint_150,v500,z100,Marcket\WObj:=wobj0;
        MoveL FDint_160,v500,z100,Marcket\WObj:=wobj0;
        MoveL FDint_170,v500,z100,Marcket\WObj:=wobj0;
        MoveL FDint_10,v500,z100,Marcket\WObj:=wobj0;

    ENDPROC
    PROC R1ext()
        MoveL GR1ext_10,v500,z100,Marcket\WObj:=wobj0;
        MoveL GR1ext_20,v500,z100,Marcket\WObj:=wobj0;
        MoveL GR1ext_30,v500,z100,Marcket\WObj:=wobj0;
        MoveL GR1ext_40,v500,z100,Marcket\WObj:=wobj0;
        MoveL GR1ext_50,v500,z100,Marcket\WObj:=wobj0;
        MoveL GR1ext_60,v500,z100,Marcket\WObj:=wobj0;
        MoveL GR1ext_70,v500,z100,Marcket\WObj:=wobj0;
        MoveL GR1ext_80,v500,z100,Marcket\WObj:=wobj0;
        MoveL GR1ext_90,v500,z100,Marcket\WObj:=wobj0;
        MoveL GR1ext_100,v500,z100,Marcket\WObj:=wobj0;
        MoveL GR1ext_110,v500,z100,Marcket\WObj:=wobj0;
        MoveL GR1ext_120,v500,z100,Marcket\WObj:=wobj0;
        MoveL GR1ext_130,v500,z100,Marcket\WObj:=wobj0;
        MoveL GR1ext_140,v500,z100,Marcket\WObj:=wobj0;
        MoveL GR1ext_150,v500,z100,Marcket\WObj:=wobj0;
        MoveL GR1ext_160,v500,z100,Marcket\WObj:=wobj0;
        MoveL GR1ext_170,v500,z100,Marcket\WObj:=wobj0;
        MoveL GR1ext_180,v500,z100,Marcket\WObj:=wobj0;
        MoveL GR1ext_190,v500,z100,Marcket\WObj:=wobj0;
        MoveL GR1ext_200,v500,z100,Marcket\WObj:=wobj0;
        MoveL GR1ext_210,v500,z100,Marcket\WObj:=wobj0;
        MoveL GR1ext_220,v500,z100,Marcket\WObj:=wobj0;
        MoveL GR1ext_230,v500,z100,Marcket\WObj:=wobj0;
        MoveL GR1ext_240,v500,z100,Marcket\WObj:=wobj0;
        MoveL GR1ext_250,v500,z100,Marcket\WObj:=wobj0;
        MoveL GR1ext_260,v500,z100,Marcket\WObj:=wobj0;
        MoveL GR1ext_270,v500,z100,Marcket\WObj:=wobj0;
        MoveL GR1ext_280,v500,z100,Marcket\WObj:=wobj0;
        MoveL GR1ext_290,v500,z100,Marcket\WObj:=wobj0;
        MoveL GR1ext_300,v500,z100,Marcket\WObj:=wobj0;
        MoveL GR1ext_310,v500,z100,Marcket\WObj:=wobj0;
        MoveL GR1ext_320,v500,z100,Marcket\WObj:=wobj0;
        MoveL GR1ext_330,v500,z100,Marcket\WObj:=wobj0;
        MoveL GR1ext_340,v500,z100,Marcket\WObj:=wobj0;
        MoveL GR1ext_350,v500,z100,Marcket\WObj:=wobj0;
        MoveL GR1ext_360,v500,z100,Marcket\WObj:=wobj0;
        MoveL GR1ext_370,v500,z100,Marcket\WObj:=wobj0;
        MoveL GR1ext_380,v500,z100,Marcket\WObj:=wobj0;
        MoveL GR1ext_390,v500,z100,Marcket\WObj:=wobj0;

    ENDPROC
    PROC R1int()
        MoveL HR1int_10,v500,z100,Marcket\WObj:=wobj0;
        MoveL HR1int_20,v500,z100,Marcket\WObj:=wobj0;
        MoveL HR1int_30,v500,z100,Marcket\WObj:=wobj0;
        MoveL HR1int_40,v500,z100,Marcket\WObj:=wobj0;
        MoveL HR1int_50,v500,z100,Marcket\WObj:=wobj0;
        MoveL HR1int_60,v500,z100,Marcket\WObj:=wobj0;
        MoveL HR1int_70,v500,z100,Marcket\WObj:=wobj0;
        MoveL HR1int_80,v500,z100,Marcket\WObj:=wobj0;
        MoveL HR1int_90,v500,z100,Marcket\WObj:=wobj0;
        MoveL HR1int_10,v500,z100,Marcket\WObj:=wobj0;

    ENDPROC
    PROC J()
        MoveL IJ_10,v500,z100,Marcket\WObj:=wobj0;
        MoveL IJ_20,v500,z100,Marcket\WObj:=wobj0;
        MoveL IJ_30,v500,z100,Marcket\WObj:=wobj0;
        MoveL IJ_40,v500,z100,Marcket\WObj:=wobj0;
        MoveL IJ_50,v500,z100,Marcket\WObj:=wobj0;
        MoveL IJ_60,v500,z100,Marcket\WObj:=wobj0;
        MoveL IJ_70,v500,z100,Marcket\WObj:=wobj0;
        MoveL IJ_80,v500,z100,Marcket\WObj:=wobj0;
        MoveL IJ_90,v500,z100,Marcket\WObj:=wobj0;
        MoveL IJ_100,v500,z100,Marcket\WObj:=wobj0;
        MoveL IJ_110,v500,z100,Marcket\WObj:=wobj0;
        MoveL IJ_120,v500,z100,Marcket\WObj:=wobj0;
        MoveL IJ_130,v500,z100,Marcket\WObj:=wobj0;
        MoveL IJ_140,v500,z100,Marcket\WObj:=wobj0;
        MoveL IJ_150,v500,z100,Marcket\WObj:=wobj0;
        MoveL IJ_160,v500,z100,Marcket\WObj:=wobj0;
        MoveL IJ_170,v500,z100,Marcket\WObj:=wobj0;
        MoveL IJ_180,v500,z100,Marcket\WObj:=wobj0;
        MoveL IJ_190,v500,z100,Marcket\WObj:=wobj0;
        MoveL IJ_200,v500,z100,Marcket\WObj:=wobj0;
        MoveL IJ_210,v500,z100,Marcket\WObj:=wobj0;
        MoveL IJ_220,v500,z100,Marcket\WObj:=wobj0;
        MoveL IJ_230,v500,z100,Marcket\WObj:=wobj0;
        MoveL IJ_240,v500,z100,Marcket\WObj:=wobj0;
        MoveL IJ_250,v500,z100,Marcket\WObj:=wobj0;
        MoveL IJ_260,v500,z100,Marcket\WObj:=wobj0;
        MoveL IJ_270,v500,z100,Marcket\WObj:=wobj0;
        MoveL IJ_280,v500,z100,Marcket\WObj:=wobj0;
        MoveL IJ_290,v500,z100,Marcket\WObj:=wobj0;
        MoveL IJ_300,v500,z100,Marcket\WObj:=wobj0;
        MoveL IJ_310,v500,z100,Marcket\WObj:=wobj0;
        MoveL IJ_320,v500,z100,Marcket\WObj:=wobj0;

    ENDPROC
    PROC R2ext()
        MoveL JR2ext_10,v500,z100,Marcket\WObj:=wobj0;
        MoveL JR2ext_20,v500,z100,Marcket\WObj:=wobj0;
        MoveL JR2ext_30,v500,z100,Marcket\WObj:=wobj0;
        MoveL JR2ext_40,v500,z100,Marcket\WObj:=wobj0;
        MoveL JR2ext_50,v500,z100,Marcket\WObj:=wobj0;
        MoveL JR2ext_60,v500,z100,Marcket\WObj:=wobj0;
        MoveL JR2ext_70,v500,z100,Marcket\WObj:=wobj0;
        MoveL JR2ext_80,v500,z100,Marcket\WObj:=wobj0;
        MoveL JR2ext_90,v500,z100,Marcket\WObj:=wobj0;
        MoveL JR2ext_100,v500,z100,Marcket\WObj:=wobj0;
        MoveL JR2ext_110,v500,z100,Marcket\WObj:=wobj0;
        MoveL JR2ext_120,v500,z100,Marcket\WObj:=wobj0;
        MoveL JR2ext_130,v500,z100,Marcket\WObj:=wobj0;
        MoveL JR2ext_140,v500,z100,Marcket\WObj:=wobj0;
        MoveL JR2ext_150,v500,z100,Marcket\WObj:=wobj0;
        MoveL JR2ext_160,v500,z100,Marcket\WObj:=wobj0;
        MoveL JR2ext_170,v500,z100,Marcket\WObj:=wobj0;
        MoveL JR2ext_180,v500,z100,Marcket\WObj:=wobj0;
        MoveL JR2ext_190,v500,z100,Marcket\WObj:=wobj0;
        MoveL JR2ext_200,v500,z100,Marcket\WObj:=wobj0;
        MoveL JR2ext_210,v500,z100,Marcket\WObj:=wobj0;
        MoveL JR2ext_220,v500,z100,Marcket\WObj:=wobj0;
        MoveL JR2ext_230,v500,z100,Marcket\WObj:=wobj0;
        MoveL JR2ext_240,v500,z100,Marcket\WObj:=wobj0;
        MoveL JR2ext_250,v500,z100,Marcket\WObj:=wobj0;
        MoveL JR2ext_260,v500,z100,Marcket\WObj:=wobj0;
        MoveL JR2ext_270,v500,z100,Marcket\WObj:=wobj0;
        MoveL JR2ext_280,v500,z100,Marcket\WObj:=wobj0;
        MoveL JR2ext_290,v500,z100,Marcket\WObj:=wobj0;
        MoveL JR2ext_300,v500,z100,Marcket\WObj:=wobj0;
        MoveL JR2ext_310,v500,z100,Marcket\WObj:=wobj0;
        MoveL JR2ext_320,v500,z100,Marcket\WObj:=wobj0;
        MoveL JR2ext_330,v500,z100,Marcket\WObj:=wobj0;
        MoveL JR2ext_340,v500,z100,Marcket\WObj:=wobj0;
        MoveL JR2ext_350,v500,z100,Marcket\WObj:=wobj0;
        MoveL JR2ext_360,v500,z100,Marcket\WObj:=wobj0;
        MoveL JR2ext_370,v500,z100,Marcket\WObj:=wobj0;
        MoveL JR2ext_380,v500,z100,Marcket\WObj:=wobj0;
        MoveL JR2ext_390,v500,z100,Marcket\WObj:=wobj0;

    ENDPROC
    PROC R2int()
        MoveL KR2int_10,v500,z100,Marcket\WObj:=wobj0;
        MoveL KR2int_20,v500,z100,Marcket\WObj:=wobj0;
        MoveL KR2int_30,v500,z100,Marcket\WObj:=wobj0;
        MoveL KR2int_40,v500,z100,Marcket\WObj:=wobj0;
        MoveL KR2int_50,v500,z100,Marcket\WObj:=wobj0;
        MoveL KR2int_60,v500,z100,Marcket\WObj:=wobj0;
        MoveL KR2int_70,v500,z100,Marcket\WObj:=wobj0;
        MoveL KR2int_80,v500,z100,Marcket\WObj:=wobj0;
        MoveL KR2int_90,v500,z100,Marcket\WObj:=wobj0;

    ENDPROC
    PROC main()
        WaitDI DI_01,1;
        SetDO DO_01,1;
        HomeToPrework;
        Renault;
        ToPreworkDR;
        Dint;
        ToPreworkDR;
        Dext;
        ToPreworkDR;
        R1int;
        ToPreworkDR;
        R1ext;
        ToPreworkDR;
        ToPreworkJR;
        J;
        ToPreworkJR;
        R2int;
        ToPreworkJR;
        R2ext;
        ToPreworkJR;
        WaitDI DI_02,1;
        SetDO DO_01,0;
        ToHome;

    ENDPROC
    PROC Renault()
        MoveL RA,v500,fine,Marcket\WObj:=wobj0;
        MoveL RB,v500,fine,Marcket\WObj:=wobj0;
        MoveL RC,v500,fine,Marcket\WObj:=wobj0;
        MoveL RD,v500,fine,Marcket\WObj:=wobj0;
        MoveL RE,v500,fine,Marcket\WObj:=wobj0;
        MoveL RF,v500,fine,Marcket\WObj:=wobj0;
        MoveL RA,v500,fine,Marcket\WObj:=wobj0;
        MoveL RH,v500,fine,Marcket\WObj:=wobj0;
        MoveL RI,v500,fine,Marcket\WObj:=wobj0;
        MoveL PreworkLogo,v500,fine,Marcket\WObj:=wobj0;
        MoveL RD,v500,fine,Marcket\WObj:=wobj0;
        MoveL RJ,v500,fine,Marcket\WObj:=wobj0;
        MoveL RG,v500,fine,Marcket\WObj:=wobj0;
        MoveL PreworkLogo,v500,fine,Marcket\WObj:=wobj0;
        MoveL RF,v500,fine,Marcket\WObj:=wobj0;
        MoveL RJ,v500,fine,Marcket\WObj:=wobj0;
        MoveL PreworkLogo,v500,fine,Marcket\WObj:=wobj0;
        MoveL RH,v500,fine,Marcket\WObj:=wobj0;
        MoveL RC,v500,fine,Marcket\WObj:=wobj0;
        MoveL PreworkLogo,v500,fine,Marcket\WObj:=wobj0;

    ENDPROC
    PROC ToPreworkDR()
        MoveL PreworkDR,v500,fine,Marcket\WObj:=wobj0;

    ENDPROC
    PROC ToPreworkJR()
        MoveL PreworkJR,v500,fine,Marcket\WObj:=wobj0;

    ENDPROC
    PROC ToHome()
        MoveL MHomeIntermed,v500,fine,Marcket\WObj:=wobj0;

    ENDPROC
ENDMODULE
